(* PLC project SmartCell.project, CODESYS CODESYS V3.5 SP22 Patch 3 *)
(* stored: creationDateTime 2026-10-03T11:56:44.8088927, modificationDateTime 2026-10-03T11:55:13.0727852 *)

PROGRAM PLC_PRG
  VAR
    tonPisca : TON;
    xLampada : BOOL;
  END_VAR

                  
tonPisca(IN := NOT tonPisca.Q, PT := T#500MS);
IF tonPisca.Q THEN
    xLampada := NOT xLampada;
END_IF
                
END_PROGRAM

CONFIGURATION Application
  RESOURCE Application ON PLC
    TASK MainTask(INTERVAL := T#20ms, PRIORITY := 1);
    PROGRAM PLC_PRG WITH MainTask : PLC_PRG;
  END_RESOURCE
END_CONFIGURATION
